Fanuc KAREL source: KB00086.KL

PROGRAM KB00086
%NOLOCKGROUP
VAR
  P1: INTEGER
  P2: INTEGER
  P3: INTEGER
  P4: INTEGER
  P5: INTEGER
  P6: INTEGER
BEGIN
  P1 = 1
  P2 = 1
  P3 = 1
  P4 = 1
  P5 = 1
  P6 = 1
  GET_POS_FRM(P1, P2, P3, P4, P5, P6)
END KB00086
